(* CoDeSys 2.3 library: file_plc.lib *)

(* Global variable list: Globale_Variablen *)
(*
 PLC1131-Library with Functions for File- and Serial-IO
 Copyright: G.Bachmann GmbH, 1998-2000, Feldkirch - Austria
*)
VAR_GLOBAL CONSTANT
	FILE_PLC_LIBVER					:	STRING(16) 	:=	'V1.40 Release';	(* Version String *)
	FILE_PLC_MMPREADY               :   BOOL        :=  TRUE;               (* MMP Ready *)

	(* Error-Return-Codes *)
	File_ERC_Ok :					DINT := 0;			(* OK *)
	File_ERC_Busy :					DINT := 1;			(* FB is busy *)
	File_ERC_Pending : 				DINT := 2;			(* FB is waiting *)
	File_ERC_Other :				DINT := -1;			(* Failure of C-function *)
	File_ERC_ParmInvalid :			DINT := -2;			(* Parameters are invalid *)
	File_ERC_PathToNothing :		DINT := -3;			(* Path is not valid (eg case sensitivity *)
	File_ERC_UncheckedPath :		DINT := -4;			(* Path has not been checked *)
	File_ERC_Already :				DINT := -5;			(* File or Dir already exists *)
	File_ERC_EndOf :				DINT := -6;			(* End of Dir reached *)
	File_ERC_NoHandle :				DINT := -7;			(* Invalid File or Dir identifier *)
	File_ERC_NoSelf :				DINT := -8;			(* Caller is no PLC *)
	File_ERC_Other2 :				DINT := -9;			(* Position- or Parameter-Set-Fail *)
	File_ERC_NoMemory :				DINT := -10;		(* Memory- or Thread-Alloc-Fail, medium is full *)
	File_ERC_Internal :				DINT := -11;		(* Internal Error 1 *)
	File_ERC_ParmInvalid2 :			DINT := -12;		(* Invalid Parameters 2 *)
	File_ERC_Internal2 :			DINT := -14;		(* Internal Error 2 *)
	File_ERC_Internal3 :			DINT := -15;		(* Internal Error 3 *)
	File_ERC_ParmInvalid3 :			DINT := -16;		(* Invalid Parameters 3 *)
	File_ERC_InvalidUse :			DINT := -17;		(* Invalid Call-Sequence or Parms *)
	File_ERC_FileIsOpen : 			DINT := -18;		(* file alreay opened *)
	File_ERC_NoFtpSupport : 		DINT := -19;		(* no FTP support for this function or FB *)
	File_ERC_InvalidFName : 		DINT := -20; 		(* specified (file)-name is not valid for its file-system *)
	File_ERC_Abort: 				DINT := -21;		(* user abort *)

	(* Constants used as 'RepairLevel' in FILE_CheckMedia() *)
	File_REPLEV_NoChange :			DINT := 0;			(* Do not repair errors *)
	File_REPLEV_CollectLost :		DINT := 1;			(* Collect lost data in new files *)
	File_REPLEV_FreeLost :			DINT := 2;			(* Free lost or damaged data *)
	File_REPLEV_DelLongNames :		DINT := 256;		(* Remove Win95 long name entries *)

	(* Constants used as 'RetCode' in FILE_BldPath() *)
	File_PATHRET_UncheckedPath :	DINT := -4;			(* Path has not been checked *)
	File_PATHRET_PathToNothing :	DINT := -3;			(* Path is not valid *)
	File_PATHRET_FilePathOk :		DINT :=  0;			(* Path is a valid dir *)
	File_PATHRET_DirPathOk : 		DINT :=  1;			(* Path is a valid file *)

	(* Constants used with FILE_FILEINFO.FileType and FILE_GtFileInfo.FileType *)
	File_TYPE_File :				DWORD := 16#8000;	(* Object to Path is File *)
	File_TYPE_Dir :					DWORD := 16#4000;	(* Object to Path is Directory *)
	File_TYPE_Mask :				DWORD := 16#F000;	(* Bits refering to Object-Type *)

	(* Constants used as 'AccessMode' in FILE_Open() and FILE_OpenSerial() *)
	File_ACCESS_RdOnly :			BYTE := 0;			(* Read-Only access *)
	File_ACCESS_WrOnly :			BYTE := 1;			(* Write-Only access *)
	File_ACCESS_RdWr :				BYTE := 2;			(* Read+Write access *)

	(* Constants used as 'OpMode' in FILE_Open() and FILE_OpenSerial() *)
	File_OPMODE_Direct :			DINT := 0;			(* Direct operation *)
	File_OPMODE_PerThread :			DINT := 1;			(* Operation by background thread *)

	(* Constants used as 'PosMode' in FILE_Open() *)
	File_POS_Rewrite :				BYTE := 0;			(* Start at 0-Position *)
	File_POS_Truncate :				BYTE := 1;			(* Truncate File to 0-Length *)
	File_POS_Append :				BYTE := 2;			(* Start at EndOfFile-Position *)
	File_POS_Create :				BYTE := 16;			(* Create File, if not existing *)

	(* Constants used as 'DataMode' in FILE_Open() *)
	File_DATA_Binary :				BYTE := 0;			(* Data in File is in Binary *)
	File_DATA_CsvREAL32 :			BYTE := 1;			(* REAL32-Values in Ascii *)
	File_DATA_CsvUINT32 :			BYTE := 2;			(* UINT32-Values in Ascii *)
	File_DATA_CsvSINT32 :			BYTE := 3;			(* SINT32-Values in Ascii *)
	File_DATA_String :				BYTE := 4;			(* Ascii-Lines as STRINGs *)

	(* Constants used as 'ParmMask' in FILE_OpenSerial() *)
	File_PARM_Options :				WORD := 16#0001;		(* use 'Options' parameter *)
	File_PARM_LineMode :			WORD := 16#0002;		(* use 'LineMode' parameter *)
	File_PARM_LineCtrl :			WORD := 16#0004;		(* use 'LineCtrl' parameter *)
	File_PARM_BaudRate :			WORD := 16#0008;		(* use 'BaudRate' parameter *)
	File_PARM_RdBufSize :			WORD := 16#0010;		(* use 'RdBufSize' parameter *)
	File_PARM_WrBufSize :			WORD := 16#0020;		(* use 'WrBufSize' parameter *)
	File_PARM_RdTimeout :			WORD := 16#0040;		(* use 'RdTimeout' parameter *)
	File_PARM_WrTimeout :			WORD := 16#0080;		(* use 'WrTimeout' parameter *)

	(* Constants used as 'Options' in FILE_OpenSerial() *)
	File_LOPTION_Raw :				DWORD := 16#00000000;	(* raw mode *)
	File_LOPTION_Echo :				DWORD := 16#00000001;	(* echo input *)
	File_LOPTION_CrMod :			DWORD := 16#00000002;	(* Translates input RETURN characters into NEWLINE; translates output NEWLINE into RETURN-LINEFEED. *)
	File_LOPTION_Tandem :			DWORD := 16#00000004;	(* ^S/^Q flow control *)
	File_LOPTION_7Bit :				DWORD := 16#00000008;	(* strip parity bit from 8 bit input *)
	File_LOPTION_MonTrap :			DWORD := 16#00000010;	(* enable trap to monitor *)
	File_LOPTION_Abort :			DWORD := 16#00000020;	(* enable shell restart *)
	File_LOPTION_Line :				DWORD := 16#00000040;	(* enable basic line protocol *)
	File_LOPTION_Terminal :			DWORD := 16#0000007F;	(* all non-raw options *)

	(* Constants used as 'LineMode' in FILE_OpenSerial() *)
	File_LMODE_Int : 				DWORD := 16#00000002;	(* COM-port in interrupt-mode *)
	File_LMODE_Task :				DWORD := 16#00000004;	(* COM-port treated by 'mSIOTASK' *)
	File_LMODE_Rs232 : 				DWORD := 16#00000000;	(* COM-port in RS232 mode *)
	File_LMODE_Rs422 :				DWORD := 16#00000010;	(* COM-port in RS422 mode *)
	File_LMODE_Rs485 :				DWORD := 16#00000020;	(* COM-port in RS485 mode *)
	File_LMODE_Tty :				DWORD := 16#00000040;	(* COM-port in 20mA mode *)
	File_LMODE_None : 				DWORD := 16#00000000;	(* COM-port no handshake *)
	File_LMODE_Hardw : 				DWORD := 16#00000100;	(* COM-port use hardware handshake *)
	File_LMODE_Softw : 				DWORD := 16#00000200; 	(* COM-port use software handshake *)
	File_LMODE_Fsafe : 				DWORD := 16#00001000;	(* COM-Port in 485 failsafe mode *)

	(* Constants used as 'LineCtrl' in FILE_OpenSerial() *)
	File_LCTRL_5Bits :				DWORD := 16#00000000;	(* 5 data bits *)
	File_LCTRL_6Bits :				DWORD := 16#00000001;	(* 6 data bits *)
	File_LCTRL_7Bits :				DWORD := 16#00000002;	(* 7 data bits *)
	File_LCTRL_8Bits :				DWORD := 16#00000003;	(* 8 data bits *)
	File_LCTRL_NoParity :			DWORD := 16#00000000;	(* no parity bit *)
	File_LCTRL_OddParity :			DWORD := 16#00000008;	(* odd parity *)
	File_LCTRL_EvenParity :			DWORD := 16#00000018;	(* even parity *)
	File_LCTRL_0Parity :			DWORD := 16#00000028;	(* parity bit always 0 *)
	File_LCTRL_1Parity :			DWORD := 16#00000038;	(* parity bit always 1 *)
	File_LCTRL_1Stop :				DWORD := 16#00000000;	(* 1 stop bit *)
	File_LCTRL_2Stop :				DWORD := 16#00000004;	(* 2 stop bits *)
	File_LCTRL_BreakOn :			DWORD := 16#00000040;	(* send of break-signal on *)
	File_LCTRL_8N1 :				DWORD := 16#00000003;	(* 8 data, no parity, 1 stop bit *)

	(* Constants used as 'Cmd' in FILE_Open() and FILE_OpenSerial() *)
	(* Flush can only be used in FB FILE_Open *)
	File_CMD_Open :					BYTE := 1;			(* open file or device *)
	File_CMD_Close :				BYTE := 2;			(* close opened file or device *)
	File_CMD_Flush :				BYTE := 3;			(* flushed data of file or device *)

	(* Constants used as 'Cmd' in FILE_DirectoryScan() *)
	File_DIRCMD_Open :				BYTE := 1;			(* open directory *)
	File_DIRCMD_Close :				BYTE := 2;			(* close opened directory *)
	File_DIRCMD_Read :				BYTE := 3;			(* read (next) entry from directory *)
	File_DIRCMD_Rewind :			BYTE := 4;			(* rewind read-position to first entry *)

	(* Constants used with File_SioModemCtrl() *)
	File_MCTRL_CTS :				DWORD := 16#00001000;	(* state of ClearToSend *)
	File_MCTRL_DSR :				DWORD := 16#00002000;	(* state of DataSetReady *)
	File_MCTRL_RI :					DWORD := 16#00004000;	(* state of RingIndicator *)
	File_MCTRL_CD :					DWORD := 16#00008000;	(* state of CarrierDetect *)
	File_MCTRL_ChangeCTS :			DWORD := 16#00000100;	(* change in ClearToSend *)
	File_MCTRL_ChangeDSR :			DWORD := 16#00000200;	(* change in DataSetReady *)
	File_MCTRL_ChangeRI :			DWORD := 16#00000400;	(* change in RingIndicator *)
	File_MCTRL_ChangeCD :			DWORD := 16#00000800;	(* change in CarrierDetect *)
	File_MCTRL_DTR :				DWORD := 16#00000001;	(* output: DataTerminalReady *)
	File_MCTRL_RTS :				DWORD := 16#00000002;	(* output: RequestToSend *)

	(* Constants used as 'CmdCode' in File_CtrlCmd() *)
	File_CTRLCMD_ModemMode :		DWORD := 16#00001100;	(* modem at serial port *)
	File_CTRLCMD_StatisticClear :	DWORD := 16#00001102;	(* clear Sio-Statistic *)
	(* + all codes for C ioctl()-function allowed (iolib.h) *)

	(* Constants for media numbers *)
	File_MEDIA_PcCard:				BYTE := 0;		(* PC-Card *)
	File_MEDIA_Ram0:				BYTE := 1;		(* Ram Disk *)
	File_MEDIA_NvRam0:				BYTE := 2;		(* CMOS RAM *)
	File_MEDIA_NvRam1:				BYTE := 3;		(* F-RAM *)
	File_MEDIA_Flash:				BYTE := 4;		(* File Flash *)
	File_MEDIA_Cfc:					BYTE := 5;		(* CF-Card *)
	File_MEDIA_UsbBulk: 			BYTE := 6;		(* MMC Drive *)
	File_MEDIA_Sd:					BYTE := 7;		(* Sd Drive *)
	File_MEDIA_Mmc: 			    BYTE := 8;		(* USB memory-stick *)
END_VAR

(* Data type *)
TYPE FILE_FILEINFO						(* return structure of File_GetFileInfo() *)
STRUCT
	RetCode : DINT;						(* success (0) - or Error-Code (<0) *)
	FileSize : UDINT;						(* Size of File in bytes *)
	FileType : DWORD;					(* Type of File/Directory (File_TYPE...) *)
	DateLastAccess : DATE_AND_TIME;	(* Date and Time of last Access *)
	DateLastModify : DATE_AND_TIME;	(* Date and Time of last Modification *)
END_STRUCT
END_TYPE

(* Data type *)
TYPE FILE_MEDIAINFO		(* return structure of File_GetMediaInfo() *)
STRUCT
	RetCode : DINT;			(* success (0) - or Error-Code (<0) *)
	WholeSize : UDINT;		(* Whole-Size of Media *)
	FreeSize : UDINT;			(* Current Free-Size of Media *)
	AutoSync : DINT;			(* AutoSync-Mode *)
END_STRUCT
END_TYPE

(* Data type *)
TYPE FILE_MEDIAINFOEX		(* return structure of File_GetMediaInfo() *)
STRUCT
	RetCode : DINT;			(* success (0) - or Error-Code (<0) *)
	WholeSizeL : UDINT;		(* Whole-Size of Media Low Byte *)
	WholeSizeH : UDINT;		(* Whole-Size of Media High Byte *)
	FreeSizeL : UDINT;		(* Current Free-Size of Media *)
	FreeSizeH : UDINT;		(* Current Free-Size of Media *)
	AutoSync : DINT;		(* AutoSync-Mode *)
END_STRUCT
END_TYPE

(* Data type *)
TYPE FILE_PATH					(* return structure of File_GetMedia() and File_BuildPath(), *)
STRUCT							(* used in many other FUNs and FBs to specify a file or dir *)
	RetCode : DINT;				(* success (0) - or Error-Code (<0) *)
	PathString : STRING(255);	(* path+name of file or directory *)
END_STRUCT
END_TYPE

(* Data type *)
(* PLC Structure of SYS_SIOINFO. For further information
	look at C-Description *)
TYPE FILE_SIOINFO :
STRUCT
	TxBusy:			BYTE; (* Tx-FIFO or shift register occupied *)
	RxBusy:			BYTE; (* Rx-FIFO or shift register occupied *)
	Spare:			ARRAY[0..1] OF BYTE; (* for alignment *)
	FifoSize:		UDINT; (* Size of FIFO in UART *)
	CycleTime:		UDINT; (* Ticks per cycle in TaskMode *)
	Variant:		UDINT; (* Variant of module *)
	Spare2:			UDINT; (* always 0 *)
END_STRUCT
END_TYPE

(* Data type *)
TYPE FILE_SIOSTATISTIC	(* return structure of File_GetSioStatistic() *)
STRUCT
	RetCode : DINT;			(* success (0) - or Error-Code (<0) *)
	RxCount : UDINT;			(* number of bytes received *)
	TxCount : UDINT;			(* number of bytes transmitted *)
	ORunErrrors : UDINT;		(* number of overrun-errors *)
	ParityErrors : UDINT;		(* number of parity-errors *)
	FrameErrors : UDINT;		(* number of frame-errors *)
	BreakInterrupts : UDINT;	(* number of break-interrupts *)
	FifoErrors : UDINT;		(* number of fifo-errors *)
	SpareField : UDINT;		(* reserved for extensions *)
END_STRUCT
END_TYPE

(* POU FILE_BldPath, ST *)
(******************************************************************************
Description: build new File-Path by appending a Name to an existing File-Path
Input:
  - ParentPath:  File-Path to append to 
  - NameToAppend:  Name to append to File-Path 
  - CheckExist:  TRUE => check if new file/dir exists 
  - Req:  request-enable 
Output:
  - Done:	TRUE => operation completed 
  - Error:	TRUE in case of error 
  - Status: 0: OK/Done, 1: BUSY, Error-Code in case of error 
  - Path: 
		FILE_PATH.RetCode : contains information on path if Input CheckExist 
							enabled, see File_PATHRET_ constants
		FILE_PATH.PathString : STRING(255) => path + name of file or directory 
							   (valid in case of success)
Return: 
  - see Output
******************************************************************************)
FUNCTION_BLOCK FILE_BldPath
VAR_INPUT
	Req: BOOL;						(* request-enable *)
	ParentPath : FILE_PATH;			(* File-Path to append to *)
	NameToAppend : STRING(31);		(* Name to append to File-Path *)
	CheckExist : BOOL;				(* TRUE => check if new file/dir exists *)
END_VAR
VAR_OUTPUT
	Path : FILE_PATH;				(* path + name of file or directory (valid in case of success) *)
	Done : BOOL;					(* TRUE => operation completed *)
	Error : BOOL;					(* TRUE in case of error *)
	Status : DINT;					(* 0: OK/Done, 1: BUSY, Error-Code in case of error *)
END_VAR
VAR
	Pltd : DWORD;
END_VAR
;
END_FUNCTION_BLOCK

(* POU FILE_BldPathEx, ST *)
(******************************************************************************
Description: build new File-Path by appending a Name to an existing File-Path. 
             Supports long filenames. 
Input:
  - ParentPath:  File-Path to append to 
  - NameToAppend:  Name to append to File-Path 
  - CheckExist:  TRUE => check if new file/dir exists 
  - Req:  request-enable 
Output:
  - Done:	TRUE => operation completed 
  - Error:	TRUE in case of error 
  - Status: 0: OK/Done, 1: BUSY, Error-Code in case of error 
  - Path: 
		FILE_PATH.RetCode : contains information on path if Input CheckExist 
							enabled, see File_PATHRET_ constants
		FILE_PATH.PathString : STRING(255) => path + name of file or directory 
							   (valid in case of success)
Return: 
  - see Output
******************************************************************************)
FUNCTION_BLOCK FILE_BldPathEx
VAR_INPUT
	Req: BOOL;						(* request-enable *)
	ParentPath : FILE_PATH;			(* File-Path to append to *)
	NameToAppend : STRING(255);		(* Name to append to File-Path *)
	CheckExist : BOOL;				(* TRUE => check if new file/dir exists *)
END_VAR
VAR_OUTPUT
	Path : FILE_PATH;				(* path + name of file or directory (valid in case of success) *)
	Done : BOOL;					(* TRUE => operation completed *)
	Error : BOOL;					(* TRUE in case of error *)
	Status : DINT;					(* 0: OK/Done, 1: BUSY, Error-Code in case of error *)
END_VAR
VAR
	Pltd : DWORD;
END_VAR
;
END_FUNCTION_BLOCK

(* POU File_BuildPath, ST *)
(******************************************************************************
Description: build new File-Path by appending a Name to an existing File-Path
Input:
  - ParentPath:  File-Path to append to 
  - NameToAppend:  Name to append to File-Path 
  - CheckExist:  TRUE => check if new file/dir exists 
  - Req:  request-enable 
Return: 
	FILE_PATH.RetCode : DINT => success (0 or 1) - or Error-Code (<0)
	FILE_PATH.PathString : STRING(255) => path+name of file or directory (valid in case of success)
******************************************************************************)
FUNCTION File_BuildPath : FILE_PATH
VAR_INPUT
	ParentPath : FILE_PATH;			(* File-Path to append to *)
	NameToAppend : STRING(31);		(* Name to append to File-Path *)
	CheckExist : BOOL;				(* TRUE => check if new file/dir exists *)
END_VAR
;
END_FUNCTION

(* POU FILE_CheckMedia, ST *)
(******************************************************************************
Description: Check/Repair file system on specified media
Input:
  - Req:  request-enable 
  - RepairLevel:  level of repair (File_REPLEV...) 
  - Media: Path which specifies media to check/repair
Output:
  - Done:  TRUE => completed, Check/Repair Ok 
  - Error:  TRUE in case of error 
  - Status:  0: OK/Done, 1: BUSY, Error-Code in case of error 
  - Media: Path which specifies media to check/repair
Return: 
  -
******************************************************************************)
FUNCTION_BLOCK FILE_CheckMedia
VAR_INPUT
	Req : BOOL;				(* request-enable *)
	RepairLevel : DINT;		(* level of repair (File_REPLEV...) *)
END_VAR
VAR_IN_OUT
	Media : FILE_PATH;		(* Path which specifies media to check/repair *)
END_VAR
VAR_OUTPUT
	Done : BOOL;			(* TRUE => completed, Check/Repair Ok *)
	Error : BOOL;			(* TRUE in case of error *)
	Status : DINT;			(* 0: OK/Done, 1: BUSY, Error-Code in case of error *)
END_VAR
VAR
	Pltd : DWORD;
END_VAR
;
END_FUNCTION_BLOCK

(* POU FILE_Copy, ST *)
(******************************************************************************
Description: Copy a file to a duplicate with another File-Path
  FTP note: Work with FTP server.
Input:
  - Req:  request-enable 
  - ReplaceExisting:  TRUE => overwrite an existing destination-file 
  - Source: original file to copy
  - Destination: specification of duplicate file 
Output:
  - Done:  TRUE => copy completed 
  - Error:  TRUE in case of error 
  - Status:  0: OK/Done, 1: BUSY, Error-Code in case of error 
  - Source: original file to copy
  - Destination: specification of duplicate file 
Return: 
  - see Output
******************************************************************************)
FUNCTION_BLOCK FILE_Copy
VAR_INPUT
	Req : BOOL;					(* request-enable *)
	ReplaceExisting : BOOL;		(* TRUE => overwrite an existing destination-file *)
END_VAR
VAR_IN_OUT
	Source : FILE_PATH;			(* original file to copy *)
	Destination : FILE_PATH;	(* specification of duplicate file *)
END_VAR
VAR_OUTPUT
	Done : BOOL;				(* TRUE => copy completed *)
	Error : BOOL;				(* TRUE in case of error *)
	Status : DINT;				(* 0: OK/Done, 1: BUSY, Error-Code in case of error *)
END_VAR
VAR
	Pltd : DWORD;
END_VAR
;
END_FUNCTION_BLOCK

(* POU FILE_CopyEx, ST *)
(******************************************************************************
Description: Copy a file to a duplicate with another File-Path
  FTP note: Work with FTP server.
Input:
  - Req:  request-enable 
  - ReplaceExisting:  TRUE => overwrite an existing destination-file 
  - Source: original file to copy
  - Destination: specification of duplicate file 
Output:
  - Done:  TRUE => copy completed 
  - Error:  TRUE in case of error 
  - Status:  0: OK/Done, 1: BUSY, Error-Code in case of error 
  - Source: original file to copy
  - Destination: specification of duplicate file 
Return: 
  - see Output
******************************************************************************)
FUNCTION_BLOCK FILE_CopyEx
VAR_INPUT
	Req : BOOL;					(* request-enable *)
	ReplaceExisting : BOOL;		(* TRUE => overwrite an existing destination-file *)
    Abort: BOOL;                (* interrupt the process *)
END_VAR
VAR_IN_OUT
	Source : FILE_PATH;			(* original file to copy *)
	Destination : FILE_PATH;	(* specification of duplicate file *)
END_VAR
VAR_OUTPUT
	Done : BOOL;				(* TRUE => copy completed *)
	Error : BOOL;				(* TRUE in case of error *)
	Status : DINT;				(* 0: OK/Done, 1: BUSY, Error-Code in case of error *)
END_VAR
VAR
	Pltd : DWORD;
END_VAR
;
END_FUNCTION_BLOCK

(* POU File_CtrlCmd, ST *)
(******************************************************************************
Description: issue a ctrl-command call (in C: ioctl()) on the specified file/device
	FTP note: A few commands are supported. See VxWorks documentation.
Input:
  - FileId:  file/device-specification to act upon 
  - CmdCode:  command-code (File_CTRLCMD...) 
  - Argument:  argument value or address 
Return: 
	DWORD => error-code (16#FFFFFFFF) or return value from driver
******************************************************************************)
FUNCTION File_CtrlCmd : DWORD
VAR_INPUT
	FileId : DWORD;			(* file/device-specification to act upon *)
	CmdCode : DWORD;		(* command-code (File_CTRLCMD...) *)
	Argument : DWORD;		(* argument value or address *)
END_VAR
;
END_FUNCTION

(* POU File_CwDirectory, ST *)
(******************************************************************************
Description: Changes the working directory.
Input:
  - WorkingDirectory: new working directory path
Return: 
	DINT => success (0) - or error (-1)
******************************************************************************)
FUNCTION File_CwDirectory : DINT
VAR_INPUT
	WorkingDirectory: FILE_PATH; (* new working directory *)
END_VAR
;
END_FUNCTION

(* POU FILE_Del, ST *)
(******************************************************************************
Description: Delete a specified file
  FTP note: Work with FTP server.
Input:
  - Req:  request-enable 
  - FileToDelete : FILE_PATH;	 path which specifies file to delete 
Output:
  - Done:  TRUE => Delete completed
  - Error:  TRUE in CASE OF error
  - Status:  0: OK/Done, 1: BUSY, Error-Code in CASE OF error
RETURN:
  - see Output
******************************************************************************)

FUNCTION_BLOCK FILE_Del
VAR_INPUT
	Req : BOOL;					(* request-enable *)
	FileToDelete : FILE_PATH;	(* path which specifies file to delete *)
END_VAR
VAR_OUTPUT
	Done : BOOL;				(* TRUE => copy completed *)
	Error : BOOL;				(* TRUE in case of error *)
	Status : DINT;				(* 0: OK/Done, 1: BUSY, Error-Code in case of error *)
END_VAR
VAR
	Pltd : DWORD;
END_VAR
;
END_FUNCTION_BLOCK

(* POU File_Delete, ST *)
(******************************************************************************
Description: Delete an existing file
  FTP note: Work with FTP server.
Input:
  - FileToDelete:  path which specifies file to delete 
Return: 
	DINT => success (0) - or error-code (<0)
******************************************************************************)
FUNCTION File_Delete : DINT
VAR_INPUT
	FileToDelete : FILE_PATH;	(* path which specifies file to delete *)
END_VAR
;
END_FUNCTION

(* POU FILE_DirectoryScan, ST *)
(******************************************************************************
Description: Scan directory for file or sub-directory entries;
  FTP note: Does not work with FTP server.
Input:
  - Req:  request-enable 
  - Cmd:  Operation-Command (File_DIRCMD...) - "open", "read", "rewind" and
    "close".
  - DirToScan: directory to scan for entries
Output:
  - Done:  TRUE => operation completed 
  - Error:  TRUE in case of error 
  - Status:  0: OK/Done, 1: BUSY, Error-Code in case of error 
  - NameFound:  name of a file or directory entry 
  - DirToScan: directory to scan for entries
Return: 
  - see Output
******************************************************************************)
FUNCTION_BLOCK FILE_DirectoryScan
VAR_INPUT
	Req : BOOL;						(* request-enable *)
	Cmd : BYTE;						(* Operation-Command (File_DIRCMD...) *)
END_VAR
VAR_IN_OUT
	DirToScan : FILE_PATH;			(* directory to scan for entries *)
END_VAR
VAR_OUTPUT
	Done : BOOL;					(* TRUE => operation completed *)
	Error : BOOL;					(* TRUE in case of error *)
	Status : DINT;					(* 0: OK/Done, 1: BUSY, Error-Code in case of error *)
	NameFound : STRING(31);			(* name of a file or directory entry *)
END_VAR
VAR
	DirId : DWORD;
END_VAR
;
END_FUNCTION_BLOCK

(* POU FILE_DirScan, ST *)
(******************************************************************************
Description: Scan directory for file or sub-directory entries.
			 Uses a background worker-task for directory-operations. 
  FTP note: Does not work with FTP server. 
Input:
  - Req:  request-enable 
  - Cmd:  Operation-Command (File_DIRCMD...) - "open", "read", "rewind" and
    "close".
  - DirToScan: directory to scan for entries
Output:
  - Done:  TRUE => operation completed 
  - Error:  TRUE in case of error 
  - Status:  0: OK/Done, 1: BUSY, Error-Code in case of error 
  - NameFound:  name of a file or directory entry
Return: 
  - see Output
******************************************************************************)
FUNCTION_BLOCK FILE_DirScan
VAR_INPUT
	Req : BOOL;					(* request-enable *)
	Cmd : BYTE;					(* Operation-Command (File_DIRCMD...) *)
	DirToScan : FILE_PATH;		(* directory to scan for entries *)
END_VAR
VAR_OUTPUT
	Done : BOOL;				(* TRUE => operation completed *)
	Error : BOOL;				(* TRUE in case of error *)
	Status : DINT;				(* 0: OK/Done, 1: BUSY, Error-Code in case of error *)
	NameFound : STRING(31);		(* name of a file or directory entry *)
END_VAR
VAR_OUTPUT
END_VAR
VAR
	Pltd : DWORD;
	DirId : DWORD;
END_VAR
;
END_FUNCTION_BLOCK

(* POU FILE_DirScanEx, ST *)
(******************************************************************************
Description: Scan directory for file or sub-directory entries.
			 Uses a background worker-task for directory-operations. 
  FTP note:  Does work with FTP server. If a hostname is given, a ftp-
			 connection with the specified host, username and password
			 is established. 
Input:
  - Req:  request-enable 
  - Cmd:  Operation-Command (File_DIRCMD...) - "open", "read" and
    "close". The "rewind" command is not supported. 
  - DirToScan: directory to scan for entries
  - Host: IP-addresse (eg "192.9.250.14") or hostname
  - User: username for authentification at the FTP-server
  - Passwd: password for authentification
Output:
  - Done:  TRUE => operation completed 
  - Error:  TRUE in case of error 
  - Status:  0: OK/Done, 1: BUSY, Error-Code in case of error 
  - NameFound:  name of a file or directory entry
Return: 
  - see Output
******************************************************************************)
FUNCTION_BLOCK FILE_DirScanEx
VAR_INPUT
	Req : BOOL;					(* request-enable *)
	Cmd : BYTE;					(* Operation-Command (File_DIRCMD...) *)
	DirToScan : FILE_PATH;		(* directory to scan for entries *)
	Host : STRING(19);			(* Hostname of FTP-server *)
	User : STRING(19);			(* Username for authentification *)
	Passwd : STRING(19);		(* Password for authentification *)
END_VAR
VAR_OUTPUT
	Done : BOOL;				(* TRUE => operation completed *)
	Error : BOOL;				(* TRUE in case of error *)
	Status : DINT;				(* 0: OK/Done, 1: BUSY, Error-Code in case of error *)
	NameFound : STRING(31);		(* name of a file or directory entry *)
END_VAR
VAR_OUTPUT
END_VAR
VAR
	Pltd : DWORD;
	DirId : DWORD;
END_VAR
;
END_FUNCTION_BLOCK

(* POU FILE_DirScanEx2, ST *)
(******************************************************************************
Description: Scan directory for file or sub-directory entries.
			 Uses a background worker-task for directory-operations. 
             Supports long filenames. 
  FTP note:  Does work with FTP server. If a hostname is given, a ftp-
			 connection with the specified host, username and password
			 is established. 
Input:
  - Req:  request-enable 
  - Cmd:  Operation-Command (File_DIRCMD...) - "open", "read" and
    "close". The "rewind" command is not supported. 
  - DirToScan: directory to scan for entries
  - Host: IP-addresse (eg "192.9.250.14") or hostname
  - User: username for authentification at the FTP-server
  - Passwd: password for authentification
Output:
  - Done:  TRUE => operation completed 
  - Error:  TRUE in case of error 
  - Status:  0: OK/Done, 1: BUSY, Error-Code in case of error 
  - NameFound:  name of a file or directory entry
Return: 
  - see Output
******************************************************************************)
FUNCTION_BLOCK FILE_DirScanEx2
VAR_INPUT
	Req : BOOL;					(* request-enable *)
	Cmd : BYTE;					(* Operation-Command (File_DIRCMD...) *)
	DirToScan : FILE_PATH;		(* directory to scan for entries *)
	Host : STRING(19);			(* Hostname of FTP-server *)
	User : STRING(19);			(* Username for authentification *)
	Passwd : STRING(19);		(* Password for authentification *)
END_VAR
VAR_OUTPUT
	Done : BOOL;				(* TRUE => operation completed *)
	Error : BOOL;				(* TRUE in case of error *)
	Status : DINT;				(* 0: OK/Done, 1: BUSY, Error-Code in case of error *)
	NameFound : STRING(255);	(* name of a file or directory entry *)
END_VAR
VAR_OUTPUT
END_VAR
VAR
	Pltd : DWORD;
	DirId : DWORD;
END_VAR
;
END_FUNCTION_BLOCK

(* POU File_Flush, ST *)
(******************************************************************************
Description: Flush all output-buffers of the specified file to the media
  FTP note: Does not work with FTP server.
Input:
  - FileId:  open file to flush buffers of 
Return: 
	DINT => success (0) - or error-code (<0)
******************************************************************************)
FUNCTION File_Flush : DINT
VAR_INPUT
	FileId : DWORD;		(* open file to flush buffers of *)
END_VAR
;
END_FUNCTION

(* POU File_GetFileInfo, ST *)
(******************************************************************************
Description: retrieve information about specified file or directory
  FTP note: Work with FTP server. DateLastAccess and DateLastModify
	are not filled correct.
Input:
  - File:  Path which specifies file/dir to get info to
Return: 
	FILE_FILEINFO.RetCode : DINT => success (0) - or Error-Code (<0)
	FILE_FILEINFO.FileSize : UDINT => Size of File in bytes
	FILE_FILEINFO.FileType : DWORD => Type of File/Directory (File_TYPE...)
	FILE_FILEINFO.DateLastAccess : DATE_AND_TIME => Date and Time of last Access
	FILE_FILEINFO.DateLastModify : DATE_AND_TIME => Date and Time of last Modification
******************************************************************************)
FUNCTION File_GetFileInfo : FILE_FILEINFO
VAR_INPUT
	File : FILE_PATH;			(* Path which specifies file/dir to get info to *)
END_VAR
;
END_FUNCTION

(* POU File_GetMedia, ST *)
(******************************************************************************
Description: retrieve starting 'File-Path' for a Media
Input:
  - MediaNum:  Media-Number (0,1,2,...) 
Return: 
	FILE_PATH.RetCode : DINT => success (0) - or Error-Code (<0)
	FILE_PATH.PathString : STRING(255) => path+name of file or directory (valid in case of success)
******************************************************************************)
FUNCTION File_GetMedia : FILE_PATH
VAR_INPUT
	MediaNum : UDINT;	(* Media-Number (0,1,2,...), see  File_MEDIA_xxx*)
END_VAR
;
END_FUNCTION

(* POU File_GetMediaInfo, ST *)
(******************************************************************************
Description: retrieve information about specified media
Input:
  - Media:  Path which specifies media to get info to 
  - FileId:  specification of open device/interface 
Return: 
	FILE_MEDIAINFO.RetCode : DINT => success (0) - or Error-Code (<0)
	FILE_MEDIAINFO.WholeSize : UDINT => Whole-Size of Media (valid in case of success)
	FILE_MEDIAINFO.FreeSize : UDINT => Current Free-Size of Media (valid in case of success)
	FILE_MEDIAINFO.AutoSync : DINT => AutoSync-Mode (valid in case of success)
******************************************************************************)
FUNCTION File_GetMediaInfo : FILE_MEDIAINFO
VAR_INPUT
	Media : FILE_PATH;			(* Path which specifies media to get info to *)
END_VAR
;
END_FUNCTION

(* POU File_GetMediaInfoEx, ST *)
(******************************************************************************
Description: retrieve information about specified media
Input:
  - Media:  Path which specifies media to get info to 
  - FileId:  specification of open device/interface 
Return: 
	FILE_MEDIAINFO.RetCode : DINT => success (0) - or Error-Code (<0)
	FILE_MEDIAINFO.WholeSizeL : UDINT => Low Byte Whole-Size of Media (valid in case of success)
	FILE_MEDIAINFO.WholeSizeH : UDINT => High Byte Whole-Size of Media (valid in case of success)
	FILE_MEDIAINFO.FreeSizeL : UDINT => Low Byte Current Free-Size of Media (valid in case of success)
	FILE_MEDIAINFO.FreeSizeH : UDINT => High Byte Current Free-Size of Media (valid in case of success)
	FILE_MEDIAINFO.AutoSync : DINT => AutoSync-Mode (valid in case of success)
******************************************************************************)
FUNCTION File_GetMediaInfoEx : FILE_MEDIAINFOEX
VAR_INPUT
	Media : FILE_PATH;			(* Path which specifies media to get info to *)
END_VAR
;
END_FUNCTION

(* POU File_GetNumOfUnread, ST *)
(******************************************************************************
Description: get number of bytes available for read in input-buffer of serial interface
Input:
  - FileId:  specification of open device/interface 
Return: 
	DINT => number of remaining bytes to read (>=0) or error-code (<0)
******************************************************************************)
FUNCTION File_GetNumOfUnread : DINT
VAR_INPUT
	FileId : DWORD;			(* specification of open device/interface *)
END_VAR
;
END_FUNCTION

(* POU File_GetNumOfWrite, ST *)
(******************************************************************************
Description: get number of bytes which are buffered for output on serial interface
Input:
  - FileId:  specification of open device/interface 
Return: 
	DINT => number of bytes waiting to be transmitted (>=0) or error-code (<0)
******************************************************************************)
FUNCTION File_GetNumOfWrite : DINT
VAR_INPUT
	FileId : DWORD;			(* specification of open device/interface *)
END_VAR
;
END_FUNCTION

(* POU File_GetSioStatistic, ST *)
(******************************************************************************
Description: retrieve statistic-information about serial-communication on serial-interface
Input:
  - FileId:  specification of open device/interface 
  - FileId:  specification of open file 
  - DirToMake:  new directory or sub-directory 
Return: 
	FILE_SIOSTATISTIC.RetCode : DINT => success (0) - or Error-Code (<0)
	FILE_SIOSTATISTIC.RxCount : UDINT => number of bytes received
	FILE_SIOSTATISTIC.TxCount : UDINT => number of bytes transmitted
	FILE_SIOSTATISTIC.ORunErrrors : UDINT => number of overrun-errors
	FILE_SIOSTATISTIC.ParityErrors : UDINT => number of parity-errors
	FILE_SIOSTATISTIC.FrameErrors : UDINT => number of frame-errors
	FILE_SIOSTATISTIC.BreakInterrupts : UDINT => number of break-interrupts
	FILE_SIOSTATISTIC.FifoErrors : UDINT => number of fifo-errors
	FILE_SIOSTATISTIC.SpareField : UDINT => reserved for extensions
******************************************************************************)
FUNCTION File_GetSioStatistic : FILE_SIOSTATISTIC
VAR_INPUT
	FileId : DWORD;		(* specification of open device/interface *)
END_VAR
;
END_FUNCTION

(* POU File_GetSize, ST *)
(******************************************************************************
Description: get the current size of a file
  FTP note: Work with FTP server.
Input:
  - FileId:  specification of open file 
Return: 
	DINT => size of file in bytes (>=0) or error-code (<0)
******************************************************************************)
FUNCTION File_GetSize : DINT
VAR_INPUT
	FileId : DWORD;		(* specification of open file *)
END_VAR
;
END_FUNCTION

(* POU File_GetVersion, ST *)
(******************************************************************************
Description: Returns the version string of the library. In simulation always
	'V1.00 Release' is returned.

Input:
	- dummy

Return: 
	Version String
******************************************************************************)
FUNCTION File_GetVersion : STRING(15)
VAR_INPUT
	dummy:	BOOL;
END_VAR
VAR
END_VAR
File_GetVersion := 'V1.00 Release';
END_FUNCTION

(* POU FILE_GtFileInfo, ST *)
(******************************************************************************
Description: retrieve information about specified file or directory
  FTP note: Work with FTP server. DateLastAccess and DateLastModify
	are not filled correct.
Input:
  - Req:  request-enable 
  - File:  Path which specifies file/dir to get info to
Output:
  - Done:	TRUE => operation completed 
  - Error:	TRUE in case of error 
  - Status: 0: OK/Done, 1: BUSY, Error-Code (<0) in case of error 
  - FileSize : UDINT => Size of File in bytes
  - FileType : DWORD => Type of File/Directory (File_TYPE...)
  - DateLastAccess : DATE_AND_TIME => Date and Time of last Access
  - DateLastModify : DATE_AND_TIME => Date and Time of last Modification
Return: 
  - see Output
******************************************************************************)
FUNCTION_BLOCK FILE_GtFileInfo
VAR_INPUT
	Req: BOOL;						(* request-enable *)
	File : FILE_PATH;				(* Path which specifies file/dir to get info to *)
END_VAR
VAR_OUTPUT
	Done : BOOL;					(* TRUE => operation completed *)
	Error : BOOL;					(* TRUE in case of error *)
	Status : DINT;					(* 0: OK/Done, 1: BUSY, Error-Code in case of error *)
	FileSize: UDINT;				(* Size of File in bytes *)
	FileType: DWORD;				(* Type of File/Directory (File_TYPE...) *)
	DateLastAccess: DATE_AND_TIME;	(* Date and Time of last Access *)
	DateLastModify: DATE_AND_TIME;	(* Date and Time of last Modification *)
END_VAR
VAR
	Pltd : DWORD;
END_VAR
;
END_FUNCTION_BLOCK

(* POU FILE_GtMediaInfo, ST *)
(******************************************************************************
Description: retrieve information about specified media
Input:
  - Req:  request-enable 
  - Media: Path which specifies media to get info to 
Output:
  - Done:	TRUE => operation completed 
  - Error:	TRUE in case of error 
  - Status: 0: OK/Done, 1: BUSY, Error-Code in case of error 
  - WholeSize : UDINT => Whole-Size of Media (valid in case of success)
  - FreeSize : UDINT => Current Free-Size of Media (valid in case of success)
  - AutoSync : DINT => AutoSync-Mode (valid in case of success)
Return: 
  - see Output
******************************************************************************)
FUNCTION_BLOCK FILE_GtMediaInfo
VAR_INPUT
	Req: BOOL;						(* request-enable *)
	Media : FILE_PATH;				(* Path which specifies media to get info to *)
END_VAR
VAR_OUTPUT
	Done : BOOL;					(* TRUE => operation completed *)
	Error : BOOL;					(* TRUE in case of error *)
	Status : DINT;					(* 0: OK/Done, 1: BUSY, Error-Code in case of error *)
	WholeSize: UDINT;				(* UDINT => Whole-Size of Media (valid in case of success) *)
	FreeSize: UDINT;				(* UDINT => Current Free-Size of Media (valid in case of success) *)
	AutoSync: DINT;					(* DINT => AutoSync-Mode (valid in case of success) *)
END_VAR
VAR
	Pltd : DWORD;
END_VAR
;
END_FUNCTION_BLOCK

(* POU FILE_GtMediaInfoEx, ST *)
(******************************************************************************
Description: retrieve information about specified media
Input:
  - Req:  request-enable 
  - Media: Path which specifies media to get info to 
Output:
  - Done:	TRUE => operation completed 
  - Error:	TRUE in case of error 
  - Status: 0: OK/Done, 1: BUSY, Error-Code in case of error 
  - WholeSizeL : UDINT => Low Byte of Whole-Size of Media (valid in case of success)
  - WholeSizeH : UDINT => High Byte of Whole-Size of Media (valid in case of success)
  - FreeSizeL : UDINT => Low Byte of Current Free-Size of Media (valid in case of success)
  - FreeSizeH : UDINT => High Byte of Current Free-Size of Media (valid in case of success)
  - AutoSync : DINT => AutoSync-Mode (valid in case of success)
Return: 
  - see Output
******************************************************************************)
FUNCTION_BLOCK FILE_GtMediaInfoEx
VAR_INPUT
	Req: BOOL;						(* request-enable *)
	Media : FILE_PATH;				(* Path which specifies media to get info to *)
END_VAR
VAR_OUTPUT
	Done : BOOL;					(* TRUE => operation completed *)
	Error : BOOL;					(* TRUE in case of error *)
	Status : DINT;					(* 0: OK/Done, 1: BUSY, Error-Code in case of error *)
	WholeSizeL: UDINT;				(* UDINT => Low Byte of Whole-Size of Media (valid in case of success) *)
	WholeSizeH: UDINT;				(* UDINT => High Byte of Whole-Size of Media (valid in case of success) *)
	FreeSizeL: UDINT;				(* UDINT => Low Byte of Current Free-Size of Media (valid in case of success) *)
	FreeSizeH: UDINT;				(* UDINT => High Byte of Current Free-Size of Media (valid in case of success) *)
	AutoSync: DINT;					(* DINT => AutoSync-Mode (valid in case of success) *)
END_VAR
VAR
	Pltd : DWORD;
END_VAR
;
END_FUNCTION_BLOCK

(* POU File_GwDirectory, ST *)
(******************************************************************************
Description: Shows the current working directory
Input:
  - BOOL dummy variable not used by File_GwDirectory internally
Return: 
	FILE_PATH containing working directory as string and error code
******************************************************************************)

FUNCTION File_GwDirectory : FILE_PATH
VAR_INPUT
	dummy: BOOL;
END_VAR
VAR
END_VAR
;
END_FUNCTION

(* POU File_IsFileNameValid, ST *)
(******************************************************************************
Description: tests if a string is a valid VxWorks file-/directoryname and 
             supplies a valid name (needs MSYS 2.10 Release or above)
Input:
  - InName: string to test
Output:
  - OutName: valid string (illegal characters are replaced with a tilde)
Return: 
  - 0  - string is a valid file-/directoryname
  - File_ERC_InvalidFName - string is not a valid file-/directoryname
******************************************************************************)
FUNCTION File_IsFileNameValid : DINT
VAR_INPUT
	InName: STRING(254);
	OutName: STRING(254);
END_VAR
VAR
END_VAR
;
END_FUNCTION

(* POU FILE_MkDir, ST *)
(******************************************************************************
Description: Create a new directory
  FTP note: Does work with FTP server.
Input:
  - DirToMake:  new directory or sub-directory 
Output:
  - Done:  TRUE => operation completed
  - Error:  TRUE in CASE OF error
  - Status:  0: OK/Done, 1: BUSY, Error-Code in CASE OF error
RETURN:
  - see Output
******************************************************************************)
FUNCTION_BLOCK FILE_MkDir
VAR_INPUT
	Req : BOOL;					(* request-enable *)
	DirToMake : FILE_PATH;		(* new directory or sub-directory *)
END_VAR
VAR_OUTPUT
	Done : BOOL;				(* TRUE => copy completed *)
	Error : BOOL;				(* TRUE in case of error *)
	Status : DINT;				(* 0: OK/Done, 1: BUSY, Error-Code in case of error *)
END_VAR
VAR
	Pltd : DWORD;
END_VAR
;
END_FUNCTION_BLOCK

(* POU File_MkDirectory, ST *)
(******************************************************************************
Description: Create a new directory
  FTP note: Does not work with FTP server.
Input:
  - DirToMake:  new directory or sub-directory 
Return: 
	DINT => success (0) - or error-code (<0)
******************************************************************************)
FUNCTION File_MkDirectory : DINT
VAR_INPUT
	DirToMake : FILE_PATH;			(* new directory or sub-directory *)
END_VAR
;
END_FUNCTION

(* POU FILE_Open, ST *)
(******************************************************************************
Description: Open a file by its path-name
  FTP note: File_CMD_Open...Work with FTP server, except of File_POS_Truncate.
            File_CMD_Close...Work with FTP server.
            File_CMD_Flush...Does not work with FTP server.
Input:
  - Req:  request-enable 
  - Cmd:  Operation-Command (File_CMD...) 
  - AccessMode:  Read/Write/RdWr (File_ACCESS...) 
  - OpMode:  Mode of operation (File_OPMODE...) 
  - PosMode:  for Write: position to start (File_POS...) 
  - DataMode:  Type of Data in file (File_DATA...) 
Output:
  - Done:  TRUE if ready 
  - Error:  TRUE in case of error 
  - Status:  0: OK/Done, 
			 1: BUSY,
			 2: pending,
			 else Error-Code in case of error 
  - FileId:  open file Identifier 
Return: 
  -
******************************************************************************)
FUNCTION_BLOCK FILE_Open
VAR_INPUT
	Req : BOOL;				(* request-enable *)
	Cmd : BYTE;				(* Operation-Command (File_CMD...) *)
	AccessMode : BYTE;		(* Read/Write/RdWr (File_ACCESS...) *)
	OpMode : DINT;			(* Mode of operation (File_OPMODE...) *)
	PosMode : BYTE;			(* for Write: position to start (File_POS...) *)
	DataMode : BYTE;		(* Type of Data in file (File_DATA...) *)
END_VAR
VAR_IN_OUT
	PathName : FILE_PATH;	(* specification of file path+name *)
END_VAR
VAR_OUTPUT
	Done : BOOL;			(* TRUE if ready *)
	Error : BOOL;			(* TRUE in case of error *)
	Status : DINT;
	FileId : DWORD;			(* open file Identifier *)
END_VAR
;
END_FUNCTION_BLOCK

(* POU FILE_OpenSerial, ST *)
(******************************************************************************
Description: Open a serial interface by CardNb / ChanNb
Input:
  - Req:  request-enable 
  - Cmd:  Operation-Command (File_CMD...) 
  - AccessMode:  Read/Write/RdWr (File_ACCESS...) 
  - OpMode:  Mode of operation (File_OPMODE...) 
  - ParmMask:  mask of bits/parameters to use (File_PARM...) 
  - Options:  Line-Options (File_LOPTION...) 
  - LineMode:  Line-Mode (File_LMODE...) 
  - LineCtrl:  Line-Control (File_LCTRL...) 
  - BaudRate:  Baud-Rate in [bd] 
  - RdBufSize:  size of input buffer 
  - WrBufSize:  size of output buffer 
  - RdTimeout:  read-timeout in [ms] 
  - WrTimeout:  write-timeout in [ms] 
  - CardNb:  Card number 
  - ChanNb:  Channel number 
Output:
  - Done:  TRUE if ready 
  - Error:  TRUE in case of error 
  - Status:  0: OK/Done, 
			 1: BUSY,
			 2: pending,
			 else Error-Code in case of error 
  - FileId:  open device/interface Identifier 
Return: 
  -
******************************************************************************)
FUNCTION_BLOCK FILE_OpenSerial
VAR_INPUT
	Req : BOOL;				(* request-enable *)
	Cmd : BYTE;				(* Operation-Command (File_CMD...) *)
	AccessMode : BYTE;		(* Read/Write/RdWr (File_ACCESS...) *)
	OpMode : DINT;			(* Mode of operation (File_OPMODE...) *)
	ParmMask : WORD;		(* mask of bits/parameters to use (File_PARM...) *)
	Options : DWORD;		(* Line-Options (File_LOPTION...) *)
	LineMode : DWORD;		(* Line-Mode (File_LMODE...) *)
	LineCtrl : DWORD;		(* Line-Control (File_LCTRL...) *)
	BaudRate : DWORD;		(* Baud-Rate in [bd] *)
	RdBufSize : WORD;		(* size of input buffer *)
	WrBufSize : WORD;		(* size of output buffer *)
	RdTimeout : WORD;		(* read-timeout in [ms] *)
	WrTimeout : WORD;		(* write-timeout in [ms] *)
	CardNb : DINT;			(* Card number *)
	ChanNb : DINT;			(* Channel number *)
END_VAR
VAR_OUTPUT
	Done : BOOL;			(* TRUE if ready *)
	Error : BOOL;			(* TRUE in case of error *)
	Status : DINT;
	FileId : DWORD;			(* open device/interface Identifier *)
END_VAR
;
END_FUNCTION_BLOCK

(* POU FILE_Read, ST *)
(******************************************************************************
Description: Read data from file. The file is given by a 'FileId' gained by a -
    and the details of operation depend on the parameters given to the -
    FILE_Open() or FILE_OpenSerial()!
  FTP note: Work with FTP server.
Input:
  - Req:  request-enable 
  - FileId:  specification of open file 
  - Addr:  address of data to be read 
  - Length:  length of data to be read 
Output:
  - Ndr:  TRUE => read completed, new data ready 
  - Error:  TRUE in case of error 
  - Status:  0: OK/Done, 1: BUSY, Error-Code in case of error 
  - NRead:  number of bytes read 
Return: 
  -
******************************************************************************)
FUNCTION_BLOCK FILE_Read
VAR_INPUT
	Req : BOOL;				(* request-enable *)
	FileId : DWORD;			(* specification of open file *)
	Addr : DWORD;			(* address of data to be read *)
	Length : UINT;			(* length of data to be read *)
END_VAR
VAR_OUTPUT
	Ndr : BOOL;				(* TRUE => read completed, new data ready *)
	Error : BOOL;			(* TRUE in case of error *)
	Status : DINT;			(* 0: OK/Done, 1: BUSY, Error-Code in case of error *)
	NRead : UINT;			(* number of bytes read *)
END_VAR
VAR
	Fi : UDINT;
END_VAR
;
END_FUNCTION_BLOCK

(* POU FILE_Ren, ST *)
(******************************************************************************
Description: Rename a file
  FTP server: Does not work with FTP server.
Input:
  - OldName:  existing file 
  - NewName:  new name for file 
  - ReplaceExisting:  TRUE => overwrite an existing file 
Output:
  - Done:  TRUE => Delete completed
  - Error:  TRUE in CASE OF error
  - Status:  0: OK/Done, 1: BUSY, Error-Code in CASE OF error
RETURN:
  - see Output
******************************************************************************)
FUNCTION_BLOCK FILE_Ren
VAR_INPUT
	Req : BOOL;					(* request-enable *)
	OldName : FILE_PATH;		(* existing file *)
	NewName : FILE_PATH;		(* new name for file *)
	ReplaceExisting : BOOL;		(* TRUE => overwrite an existing file *)
END_VAR
VAR_OUTPUT
	Done : BOOL;				(* TRUE => copy completed *)
	Error : BOOL;				(* TRUE in case of error *)
	Status : DINT;				(* 0: OK/Done, 1: BUSY, Error-Code in case of error *)
END_VAR
VAR
	Pltd : DWORD;
END_VAR
;
END_FUNCTION_BLOCK

(* POU File_Rename, ST *)
(******************************************************************************
Description: Rename a file
  FTP server: Does not work with FTP server.
Input:
  - OldName:  existing file 
  - NewName:  new name for file 
  - ReplaceExisting:  TRUE => overwrite an existing file 
Return: 
	DINT => success (0) - or error-code (<0)
******************************************************************************)
FUNCTION File_Rename : DINT
VAR_INPUT
	OldName : FILE_PATH;			(* existing file *)
	NewName : FILE_PATH;			(* new name for file *)
	ReplaceExisting : BOOL;			(* TRUE => overwrite an existing file *)
END_VAR
;
END_FUNCTION

(* POU FILE_RmDir, ST *)
(******************************************************************************
Description: Delete an existing empty directory
  FTP note: Does not work with FTP server.
Input:
  - DirToRemove:  directory to delete 
Output:
  - Done:  TRUE => Delete completed
  - Error:  TRUE in CASE OF error
  - Status:  0: OK/Done, 1: BUSY, Error-Code in CASE OF error
RETURN:
  - see Output
******************************************************************************)
FUNCTION_BLOCK FILE_RmDir
VAR_INPUT
	Req : BOOL;					(* request-enable *)
	DirToRemove: FILE_PATH;		(* directory to delete *)
END_VAR
VAR_OUTPUT
	Done : BOOL;				(* TRUE => copy completed *)
	Error : BOOL;				(* TRUE in case of error *)
	Status : DINT;				(* 0: OK/Done, 1: BUSY, Error-Code in case of error *)
END_VAR
VAR
	Pltd : DWORD;
END_VAR
;
END_FUNCTION_BLOCK

(* POU File_RmDirectory, ST *)
(******************************************************************************
Description: Delete an existing empty directory
  FTP note: Does not work with FTP server.
Input:
  - DirToRemove:  directory to delete 
Return: 
	DINT => success (0) - or error-code (<0)
******************************************************************************)
FUNCTION File_RmDirectory : DINT
VAR_INPUT
	DirToRemove: FILE_PATH;		(* directory to delete *)
END_VAR
;
END_FUNCTION

(* POU File_Seek, ST *)
(******************************************************************************
Description: set read/write-pointer in file to specified position
  FTP note: Work with FTP server.
Input:
  - FileId:  specification of open file 
  - Position:  new read/write-position 
Return: 
	DINT => success (0) or error-code (<0)
******************************************************************************)
FUNCTION File_Seek : DINT
VAR_INPUT
	FileId : DWORD;			(* specification of open file *)
	Position: DINT;			(* new read/write-position *)
END_VAR
;
END_FUNCTION

(* POU File_SioCancel, ST *)
(******************************************************************************
Description: cancel read/write operations on specified interface by clearing
    input/output-buffers
Input:
  - FileId:  specification of open device/interface 
  - CancelRead:  cancel read-operation 
  - CancelWrite:  cancel write-operation 
Return: 
	DINT => success (0) - or error-code (<0)
******************************************************************************)
FUNCTION File_SioCancel : DINT
VAR_INPUT
	FileId : DWORD;			(* specification of open device/interface *)
	CancelRead : BOOL;		(* cancel read-operation *)
	CancelWrite : BOOL;		(* cancel write-operation *)
END_VAR
;
END_FUNCTION

(* POU File_SioInfoGet, ST *)
(******************************************************************************
Description: Get Info of Device. For futher information see SIO_INFO_GET in
	C-Descrition.

Input:
  - FileId:  specification of open device/interface 

Return: 
	Filled FILE_SIOINFO	Info structure. 
	Attention: No infomation if function call fails.
******************************************************************************)

FUNCTION File_SioInfoGet : FILE_SIOINFO
VAR_INPUT
	FileId : DWORD;			(* specification of open device/interface *)
END_VAR
VAR
END_VAR
;
END_FUNCTION

(* POU File_SioLineGet, ST *)
(******************************************************************************
Description: Get line Mode bits of the device. For further Information see
	SIO_xxx definitions in msys_e.h.

Input:
  - FileId:  specification of open device/interface 

Return: 
	<0...Function call failed (see File_ERC_xxx)
	else...Mask of bits of the device
******************************************************************************)
FUNCTION File_SioLineGet : DINT
VAR_INPUT
	FileId : DWORD;			(* specification of open device/interface *)
END_VAR
VAR
END_VAR
File_SioLineGet := 0;
END_FUNCTION

(* POU File_SioLineSet, ST *)
(******************************************************************************
Description: Set line Mode bits of the device. For further Information see
	SIO_xxx definitions in msys_e.h.

Input:
  - FileId:  specification of open device/interface 
  - ModeMask: Mask of the of the device 

Return: 
	0...OK
	<0...Function call failed (see File_ERC_xxx)
******************************************************************************)
FUNCTION File_SioLineSet : DINT
VAR_INPUT
	ModeMask:	DWORD;
	FileId: 	DWORD;			(* specification of open device/interface *)
END_VAR
VAR
END_VAR
;
END_FUNCTION

(* POU File_SioModemCtrl, ST *)
(******************************************************************************
Description: modify modem-ctrl signal of the specified serial interface
Input:
  - FileId:  specification of open device/interface 
  - ValidMask:  mask of bits/signals to treat (used with Set and Get!) 
  - ValueMask:  value of bits/signals to set to (File_MCTRL...) 
  - Modify:  TRUE => Set signals, else only Get 
Return: 
	DINT => error-code (16#FFFFFFFF) or state of the signals (before 
			modify of the function itself) 
******************************************************************************)
FUNCTION File_SioModemCtrl : DWORD
VAR_INPUT
	FileId : DWORD;		(* specification of open device/interface *)
	ValidMask : DWORD;	(* mask of bits/signals to treat (used with Set and Get!) *)
	ValueMask : DWORD;	(* value of bits/signals to set to (File_MCTRL...) *)
	Modify : BOOL;		(* TRUE => Set signals, else only Get *)
END_VAR
;
END_FUNCTION

(* POU File_Tell, ST *)
(******************************************************************************
Description: get the current position of the read/write-pointer of the file
  FTP note: Work with FTP server.
Input:
  - FileId:  specification of open file 
Return: 
	DINT => position-value (>=0) or error-code (<0)
******************************************************************************)
FUNCTION File_Tell : DINT
VAR_INPUT
	FileId : DWORD;		(* specification of open file *)
END_VAR
;
END_FUNCTION

(* POU File_UnzipFile, ST *)
(******************************************************************************
Description: Extracts a ZIP archive to a folder. 
FTP note: Does not work with FTP server.
Input:
  - Req:  request-enable 
  - ZipFileName: name of the ZIP archive
  - Destination: destination path
  - ExtractWithoutPath: flag for extraction without or with zipped pathes
Output:
  - Status:  0: OK/Done, 1: BUSY, Error-Code in case of error 
Return: 
  -
******************************************************************************)
FUNCTION_BLOCK File_UnzipFile
VAR
	Pltd: DWORD;
END_VAR
VAR_INPUT
	Req: BOOL; (* request-enable *)
	ZipFileName: FILE_PATH; (* path + name of zip file *)
	Destination: FILE_PATH; (* destination path *)
	ExtractWithoutPath: BOOL; (* flag for extraction without or with zipped pathes *)
END_VAR
VAR_OUTPUT
	Done: BOOL; (* TRUE => Unzip completed *)
	Error: BOOL; (* TRUE in case of error *)
	Status: DINT; (* 0: OK/Done, 1: BUSY, Error-Code in case of error *)
END_VAR
;
END_FUNCTION_BLOCK

(* POU FILE_Write, ST *)
(******************************************************************************
Description: Write to file; the file is given by a 'FileId' gained by a
    and the details of operation depend on the parameters given to the 
    FILE_Open() or FILE_OpenSerial()!
  FTP note: Work with FTP server.
Input:
  - Req:  request-enable 
  - FileId:  specification of open file 
  - Addr:  address of data to be written 
  - Length:  length of data to be written 
Output:
  - Done:  TRUE => write completed 
  - Error:  TRUE in case of error 
  - Status:  0: OK/Done, 1: BUSY, Error-Code in case of error 
  - NWritten:  number of bytes written 
Return: 
  -
******************************************************************************)
FUNCTION_BLOCK FILE_Write
VAR_INPUT
	Req : BOOL;				(* request-enable *)
	FileId : DWORD;			(* specification of open file *)
	Addr : DWORD;			(* address of data to be written *)
	Length : UINT;			(* length of data to be written *)
END_VAR
VAR_OUTPUT
	Done : BOOL;			(* TRUE => write completed *)
	Error : BOOL;			(* TRUE in case of error *)
	Status : DINT;			(* 0: OK/Done, 1: BUSY, Error-Code in case of error *)
	NWritten : UINT;		(* number of bytes written *)
END_VAR
VAR
	Pltd : DWORD;
	Fi : UDINT;
END_VAR
;
END_FUNCTION_BLOCK

(* POU File_ZipDirectory, ST *)
(******************************************************************************
Description: Compresses a directory to a ZIP archive. It doesn't include 
	     subdirectories.
FTP note: Does not work with FTP server.
Input:
  - Req:  request-enable 
  - Directory:   directory which has to be zipped
  - ZipFileName: name of the ZIP archive
  - PackWithoutPath: flag for compression with or without path in zip archive
Output:
  - Status:  0: OK/Done, 1: BUSY, Error-Code in case of error 
Return: 
  -
******************************************************************************)
FUNCTION_BLOCK File_ZipDirectory
VAR
	Pltd: DWORD;
END_VAR
VAR_INPUT
	Req: BOOL; (* request-enable *)
	Directory: FILE_PATH; (* Path/Name of directory which has to be zipped *)
	ZipFileName: FILE_PATH; (* Name of the zip archive *)
	PackWithoutPath: BOOL; (* flag for compression with or without path in zip archive *)
END_VAR
VAR_OUTPUT
	Done: BOOL; (* TRUE => write completed *)
	Error: BOOL; (* TRUE in case of error *)
	Status: DINT; (* 0: OK/Done, 1: BUSY, Error-Code in case of error *)
END_VAR
;
END_FUNCTION_BLOCK

(* POU File_ZipFile, ST *)
(******************************************************************************
Description: Compresses a file to a ZIP archive.
FTP note: Does not work with FTP server.
Input:
  - Req:  request-enable 
  - File:   file which has to be zipped
  - ZipFileName: name of the ZIP archive
Output:
  - Status:  0: OK/Done, 1: BUSY, Error-Code in case of error 
Return: 
  -
******************************************************************************)
FUNCTION_BLOCK File_ZipFile
VAR
	Pltd: DWORD;
END_VAR
VAR_INPUT
	Req: BOOL; (* request-enable *)
	File: FILE_PATH; (* Path/Name of file which has to be zipped *)
	ZipFileName: FILE_PATH; (* Name of the zip archive *)
END_VAR
VAR_OUTPUT
	Done: BOOL; (* TRUE => write completed *)
	Error: BOOL; (* TRUE in case of error *)
	Status: DINT; (* 0: OK/Done, 1: BUSY, Error-Code in case of error *)
END_VAR
;
END_FUNCTION_BLOCK
